FUNCTION_BLOCK FB_Sensor_OMRON_E3AS EXTENDS FB_BaseDevice
VAR
	bRawInputNO AT %I*: BOOL;
	bRawInputNC AT %I*: BOOL;
END_VAR

IF bRawInputNO AND (NOT bRawInputNC) THEN			// add some cross-checking with timers in here to detect failure of contacts
	eState := E_DeviceState.ON;
ELSIF (NOT bRawInputNO) AND bRawInputNC THEN
	eState := E_DeviceState.OFF;
END_IF

END_FUNCTION_BLOCK

(* stored: Version 1.1.0.1, ProductVersion 3.1.4024.12
   POU FB_Sensor_OMRON_E3AS: Id {dba06728-3d94-4547-8c6c-4e315caf6db6}, SpecialFunc None *)
